{attribute 'qualified_only'}
{attribute 'strict'}
TYPE E_LeakTestState :
(
	IDLE := 0,
	PRESSURE_UP := 1,
	HOLD_PRESSURE :=2
);
END_TYPE

(* stored: Version 1.1.0.1, ProductVersion 3.1.4024.15
   DUT E_LeakTestState: Id {0f980a77-59b5-45f8-94e0-2fdd5c585d80} *)
